{attribute addProperty BoxType "EL3692-0000-0017"}
{attribute addProperty Id "SAI_Inputs_Channel_1AT %I*SAI_Inputs_Channel_64E745974860SAI_Range_Channel_1AT %I*SAI_Range_Channel_DF9848341620SAI_Inputs_Real_Channel_1AT %I*SAI_Inputs_Real_Channel_5F0304D13240SAI_Inputs_Channel_2AT %I*SAI_Inputs_Channel_64E745974860SAI_Range_Channel_2AT %I*SAI_Range_Channel_DF9848341620SAI_Inputs_Real_Channel_2AT %I*SAI_Inputs_Real_Channel_5F0304D13240WcStateAT %I*WcState_F855686C1620InfoDataAT %I*InfoData_BC63D37F80100"}
{attribute addProperty CRC "659662888"}
{attribute addProperty SizeInBites "288"}
{attribute addProperty SizeInBytes "36"}
TYPE EL3692_E9B845C4 :
STRUCT
	{attribute addProperty Name "SAI_Inputs_Channel_1"}
	SAI_Inputs_Channel_1 : SAI_Inputs_Channel_64E74597;
	{attribute addProperty Name "SAI_Range_Channel_1"}
	SAI_Range_Channel_1 : SAI_Range_Channel_DF984834;
	{attribute addProperty Name "SAI_Inputs_Real_Channel_1"}
	SAI_Inputs_Real_Channel_1 : SAI_Inputs_Real_Channel_5F0304D1;
	{attribute addProperty Name "SAI_Inputs_Channel_2"}
	SAI_Inputs_Channel_2 : SAI_Inputs_Channel_64E74597;
	{attribute addProperty Name "SAI_Range_Channel_2"}
	SAI_Range_Channel_2 : SAI_Range_Channel_DF984834;
	{attribute addProperty Name "SAI_Inputs_Real_Channel_2"}
	SAI_Inputs_Real_Channel_2 : SAI_Inputs_Real_Channel_5F0304D1;
	{attribute addProperty Name "WcState"}
	WcState : WcState_F855686C;
	{attribute addProperty Name "InfoData"}
	InfoData : InfoData_BC63D37F;
END_STRUCT
END_TYPE

(* stored: Version 1.2.0.0, ProductVersion 3.1.4024.9
   DUT EL3692_E9B845C4: Id {1f7785bc-a722-4968-b0ba-dd2dd285689b} *)
